{attribute addProperty BoxType "EL6201-0000-0017"}
{attribute addProperty Id "Slave_24A_DO0BIT10.125185Slave_24A_DO1BIT10.125186Slave_24A_DO2BIT10.125187Slave_24A_DO3BIT10.125188Slave_24B_DO0BIT10.125189Slave_24B_DO1BIT10.125190Slave_24B_DO2BIT10.125191Slave_24B_DO3BIT10.125192"}
{attribute addProperty CRC "1591853563"}
{attribute addProperty SizeInBites "8"}
{attribute addProperty SizeInBytes "1"}
TYPE Slave_24_Outputs_5EE1C1FB :
STRUCT
	{attribute addProperty Name "Slave_24A_DO0"}
	Slave_24A_DO0 : BIT;
	{attribute addProperty Name "Slave_24A_DO1"}
	Slave_24A_DO1 : BIT;
	{attribute addProperty Name "Slave_24A_DO2"}
	Slave_24A_DO2 : BIT;
	{attribute addProperty Name "Slave_24A_DO3"}
	Slave_24A_DO3 : BIT;
	{attribute addProperty Name "Slave_24B_DO0"}
	Slave_24B_DO0 : BIT;
	{attribute addProperty Name "Slave_24B_DO1"}
	Slave_24B_DO1 : BIT;
	{attribute addProperty Name "Slave_24B_DO2"}
	Slave_24B_DO2 : BIT;
	{attribute addProperty Name "Slave_24B_DO3"}
	Slave_24B_DO3 : BIT;
END_STRUCT
END_TYPE

(* stored: Version 1.2.0.0, ProductVersion 3.1.4024.9
   DUT Slave_24_Outputs_5EE1C1FB: Id {3592c122-5a4c-4bdb-8e70-3dff8b9e1e7b} *)
